Staubli VAL3: Day3.dtx

mdesc mNomSpeed
string sInput
num nInput
lists lResult
  [0]
    string sString
string sCommand
num nValue
string sValue
lists_num lLists_num = {}
num nNum
num nSumPerCol
num nBitResult[12]
num nBitGamma[12]
num nBitEpsilon[12]
num nEpsilon
num nGamma
num nResult
num nDeleteIndex
num nBitOxygen[12]
num nBitCO2[12]
num nResult2
